VAR_GLOBAL
	bButton 	AT %I* :BOOL;
	
	
	bGreenLight		AT %Q*: BOOL;
	bRedLight		AT %Q*: BOOL;
END_VAR

(* stored: Version 1.1.0.1, ProductVersion 3.1.4018.5
   GVL GVL: Id {38cac7d3-aa46-45eb-911e-aeaa0889797a} *)
